SYSTEM temexdmodluyben2
  (* Version 1.0, Author, 4DIAC-Consortium *)
  APPLICATION temexdmod
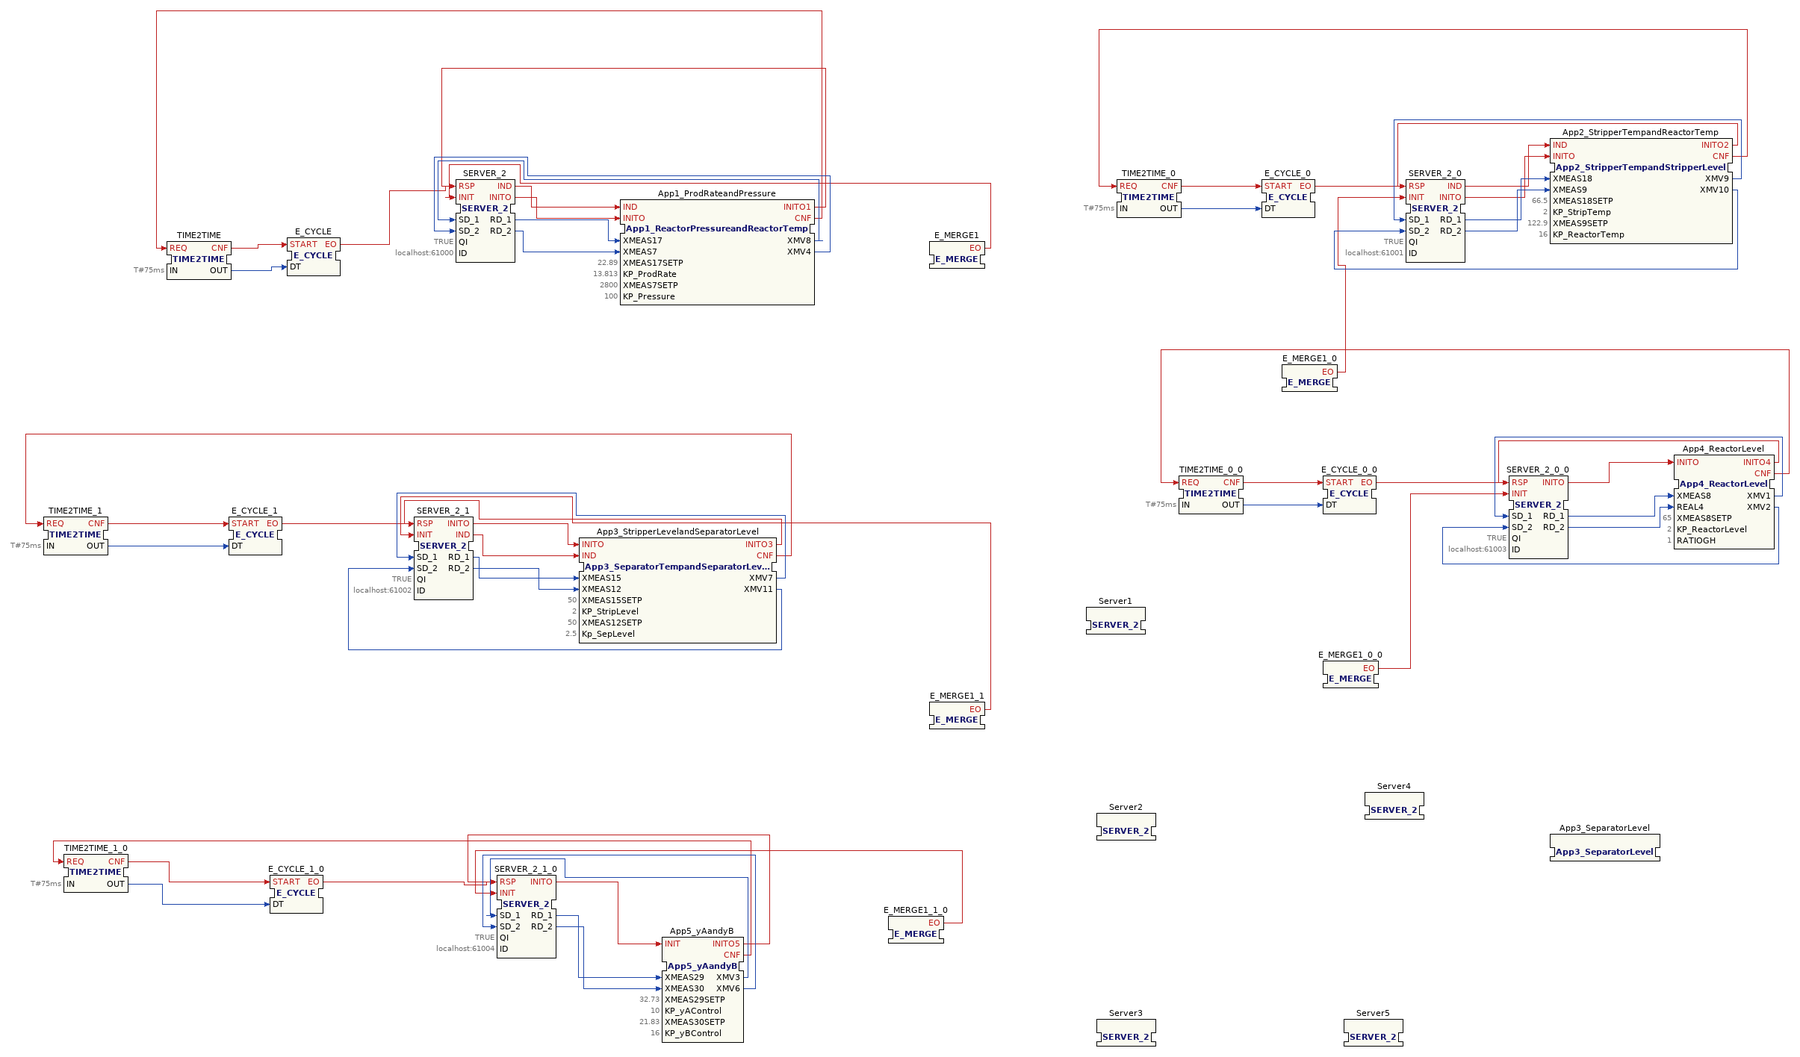
    FBS
      E_MERGE1 : E_MERGE;
      SERVER_2 : SERVER_2(QI := TRUE, ID := localhost:61000);
      TIME2TIME : TIME2TIME(IN := T#75ms);
      E_CYCLE : E_CYCLE;
      App1_ProdRateandPressure : App1_ReactorPressureandReactorTemp(XMEAS17SETP := 22.89, KP_ProdRate := 13.813, XMEAS7SETP := 2800, KP_Pressure := 100);
      TIME2TIME_0 : TIME2TIME(IN := T#75ms);
      E_CYCLE_0 : E_CYCLE;
      SERVER_2_0 : SERVER_2(QI := TRUE, ID := localhost:61001);
      E_MERGE1_0 : E_MERGE;
      App2_StripperTempandReactorTemp : App2_StripperTempandStripperLevel(XMEAS18SETP := 66.5, KP_StripTemp := 2, XMEAS9SETP := 122.9, KP_ReactorTemp := 16);
      App3_StripperLevelandSeparatorLevel : App3_SeparatorTempandSeparatorLevel(XMEAS15SETP := 50, KP_StripLevel := 2, XMEAS12SETP := 50, Kp_SepLevel := 2.5);
      SERVER_2_1 : SERVER_2(QI := TRUE, ID := localhost:61002);
      E_CYCLE_1 : E_CYCLE;
      TIME2TIME_1 : TIME2TIME(IN := T#75ms);
      E_MERGE1_1 : E_MERGE;
      App4_ReactorLevel : App4_ReactorLevel(XMEAS8SETP := 65, KP_ReactorLevel := 2, RATIOGH := 1);
      TIME2TIME_0_0 : TIME2TIME(IN := T#75ms);
      E_CYCLE_0_0 : E_CYCLE;
      SERVER_2_0_0 : SERVER_2(QI := TRUE, ID := localhost:61003);
      E_MERGE1_0_0 : E_MERGE;
      App5_yAandyB : App5_yAandyB(XMEAS29SETP := 32.73, KP_yAControl := 10, XMEAS30SETP := 21.83, KP_yBControl := 16);
      E_CYCLE_1_0 : E_CYCLE;
      SERVER_2_1_0 : SERVER_2(QI := TRUE, ID := localhost:61004);
      TIME2TIME_1_0 : TIME2TIME(IN := T#75ms);
      E_MERGE1_1_0 : E_MERGE;
      Server1 : SERVER_2;
      Server2 : SERVER_2;
      Server3 : SERVER_2;
      Server4 : SERVER_2;
      Server5 : SERVER_2;
      App3_SeparatorLevel : App3_SeparatorLevel;
    END_FBS
    EVENT_CONNECTIONS
      App1_ProdRateandPressure.INITO1 TO SERVER_2.RSP;
      SERVER_2.IND TO App1_ProdRateandPressure.IND;
      SERVER_2.INITO TO App1_ProdRateandPressure.INITO;
      TIME2TIME.CNF TO E_CYCLE.START;
      E_CYCLE.EO TO SERVER_2.RSP;
      App1_ProdRateandPressure.CNF TO TIME2TIME.REQ;
      E_MERGE1.EO TO SERVER_2.INIT;
      TIME2TIME_0.CNF TO E_CYCLE_0.START;
      E_CYCLE_0.EO TO SERVER_2_0.RSP;
      E_MERGE1_0.EO TO SERVER_2_0.INIT;
      SERVER_2_0.IND TO App2_StripperTempandReactorTemp.IND;
      SERVER_2_0.INITO TO App2_StripperTempandReactorTemp.INITO;
      App2_StripperTempandReactorTemp.INITO2 TO SERVER_2_0.RSP;
      App2_StripperTempandReactorTemp.CNF TO TIME2TIME_0.REQ;
      TIME2TIME_1.CNF TO E_CYCLE_1.START;
      E_CYCLE_1.EO TO SERVER_2_1.RSP;
      SERVER_2_1.INITO TO App3_StripperLevelandSeparatorLevel.INITO;
      SERVER_2_1.IND TO App3_StripperLevelandSeparatorLevel.IND;
      App3_StripperLevelandSeparatorLevel.INITO3 TO SERVER_2_1.RSP;
      App3_StripperLevelandSeparatorLevel.CNF TO TIME2TIME_1.REQ;
      E_MERGE1_1.EO TO SERVER_2_1.INIT;
      TIME2TIME_0_0.CNF TO E_CYCLE_0_0.START;
      E_CYCLE_0_0.EO TO SERVER_2_0_0.RSP;
      SERVER_2_0_0.INITO TO App4_ReactorLevel.INITO;
      App4_ReactorLevel.INITO4 TO SERVER_2_0_0.RSP;
      App4_ReactorLevel.CNF TO TIME2TIME_0_0.REQ;
      E_MERGE1_0_0.EO TO SERVER_2_0_0.INIT;
      SERVER_2_1_0.INITO TO App5_yAandyB.INIT;
      App5_yAandyB.INITO5 TO SERVER_2_1_0.RSP;
      App5_yAandyB.CNF TO TIME2TIME_1_0.REQ;
      TIME2TIME_1_0.CNF TO E_CYCLE_1_0.START;
      E_CYCLE_1_0.EO TO SERVER_2_1_0.RSP;
      E_MERGE1_1_0.EO TO SERVER_2_1_0.INIT;
    END_CONNECTIONS
    DATA_CONNECTIONS
      SERVER_2.RD_1 TO App1_ProdRateandPressure.XMEAS17;
      SERVER_2.RD_2 TO App1_ProdRateandPressure.XMEAS7;
      App1_ProdRateandPressure.XMV8 TO SERVER_2.SD_1;
      App1_ProdRateandPressure.XMV4 TO SERVER_2.SD_2;
      TIME2TIME.OUT TO E_CYCLE.DT;
      SERVER_2_0.RD_1 TO App2_StripperTempandReactorTemp.XMEAS18;
      SERVER_2_0.RD_2 TO App2_StripperTempandReactorTemp.XMEAS9;
      App2_StripperTempandReactorTemp.XMV9 TO SERVER_2_0.SD_1;
      App2_StripperTempandReactorTemp.XMV10 TO SERVER_2_0.SD_2;
      TIME2TIME_0.OUT TO E_CYCLE_0.DT;
      TIME2TIME_1.OUT TO E_CYCLE_1.DT;
      SERVER_2_1.RD_1 TO App3_StripperLevelandSeparatorLevel.XMEAS15;
      SERVER_2_1.RD_2 TO App3_StripperLevelandSeparatorLevel.XMEAS12;
      App3_StripperLevelandSeparatorLevel.XMV7 TO SERVER_2_1.SD_1;
      App3_StripperLevelandSeparatorLevel.XMV11 TO SERVER_2_1.SD_2;
      TIME2TIME_0_0.OUT TO E_CYCLE_0_0.DT;
      SERVER_2_0_0.RD_1 TO App4_ReactorLevel.XMEAS8;
      SERVER_2_0_0.RD_2 TO App4_ReactorLevel.REAL4;
      App4_ReactorLevel.XMV1 TO SERVER_2_0_0.SD_1;
      App4_ReactorLevel.XMV2 TO SERVER_2_0_0.SD_2;
      TIME2TIME_1_0.OUT TO E_CYCLE_1_0.DT;
      SERVER_2_1_0.RD_1 TO App5_yAandyB.XMEAS29;
      SERVER_2_1_0.RD_2 TO App5_yAandyB.XMEAS30;
      App5_yAandyB.XMV3 TO SERVER_2_1_0.SD_1;
      App5_yAandyB.XMV6 TO SERVER_2_1_0.SD_2;
    END_CONNECTIONS
  END_APPLICATION
  APPLICATION temexdmod2
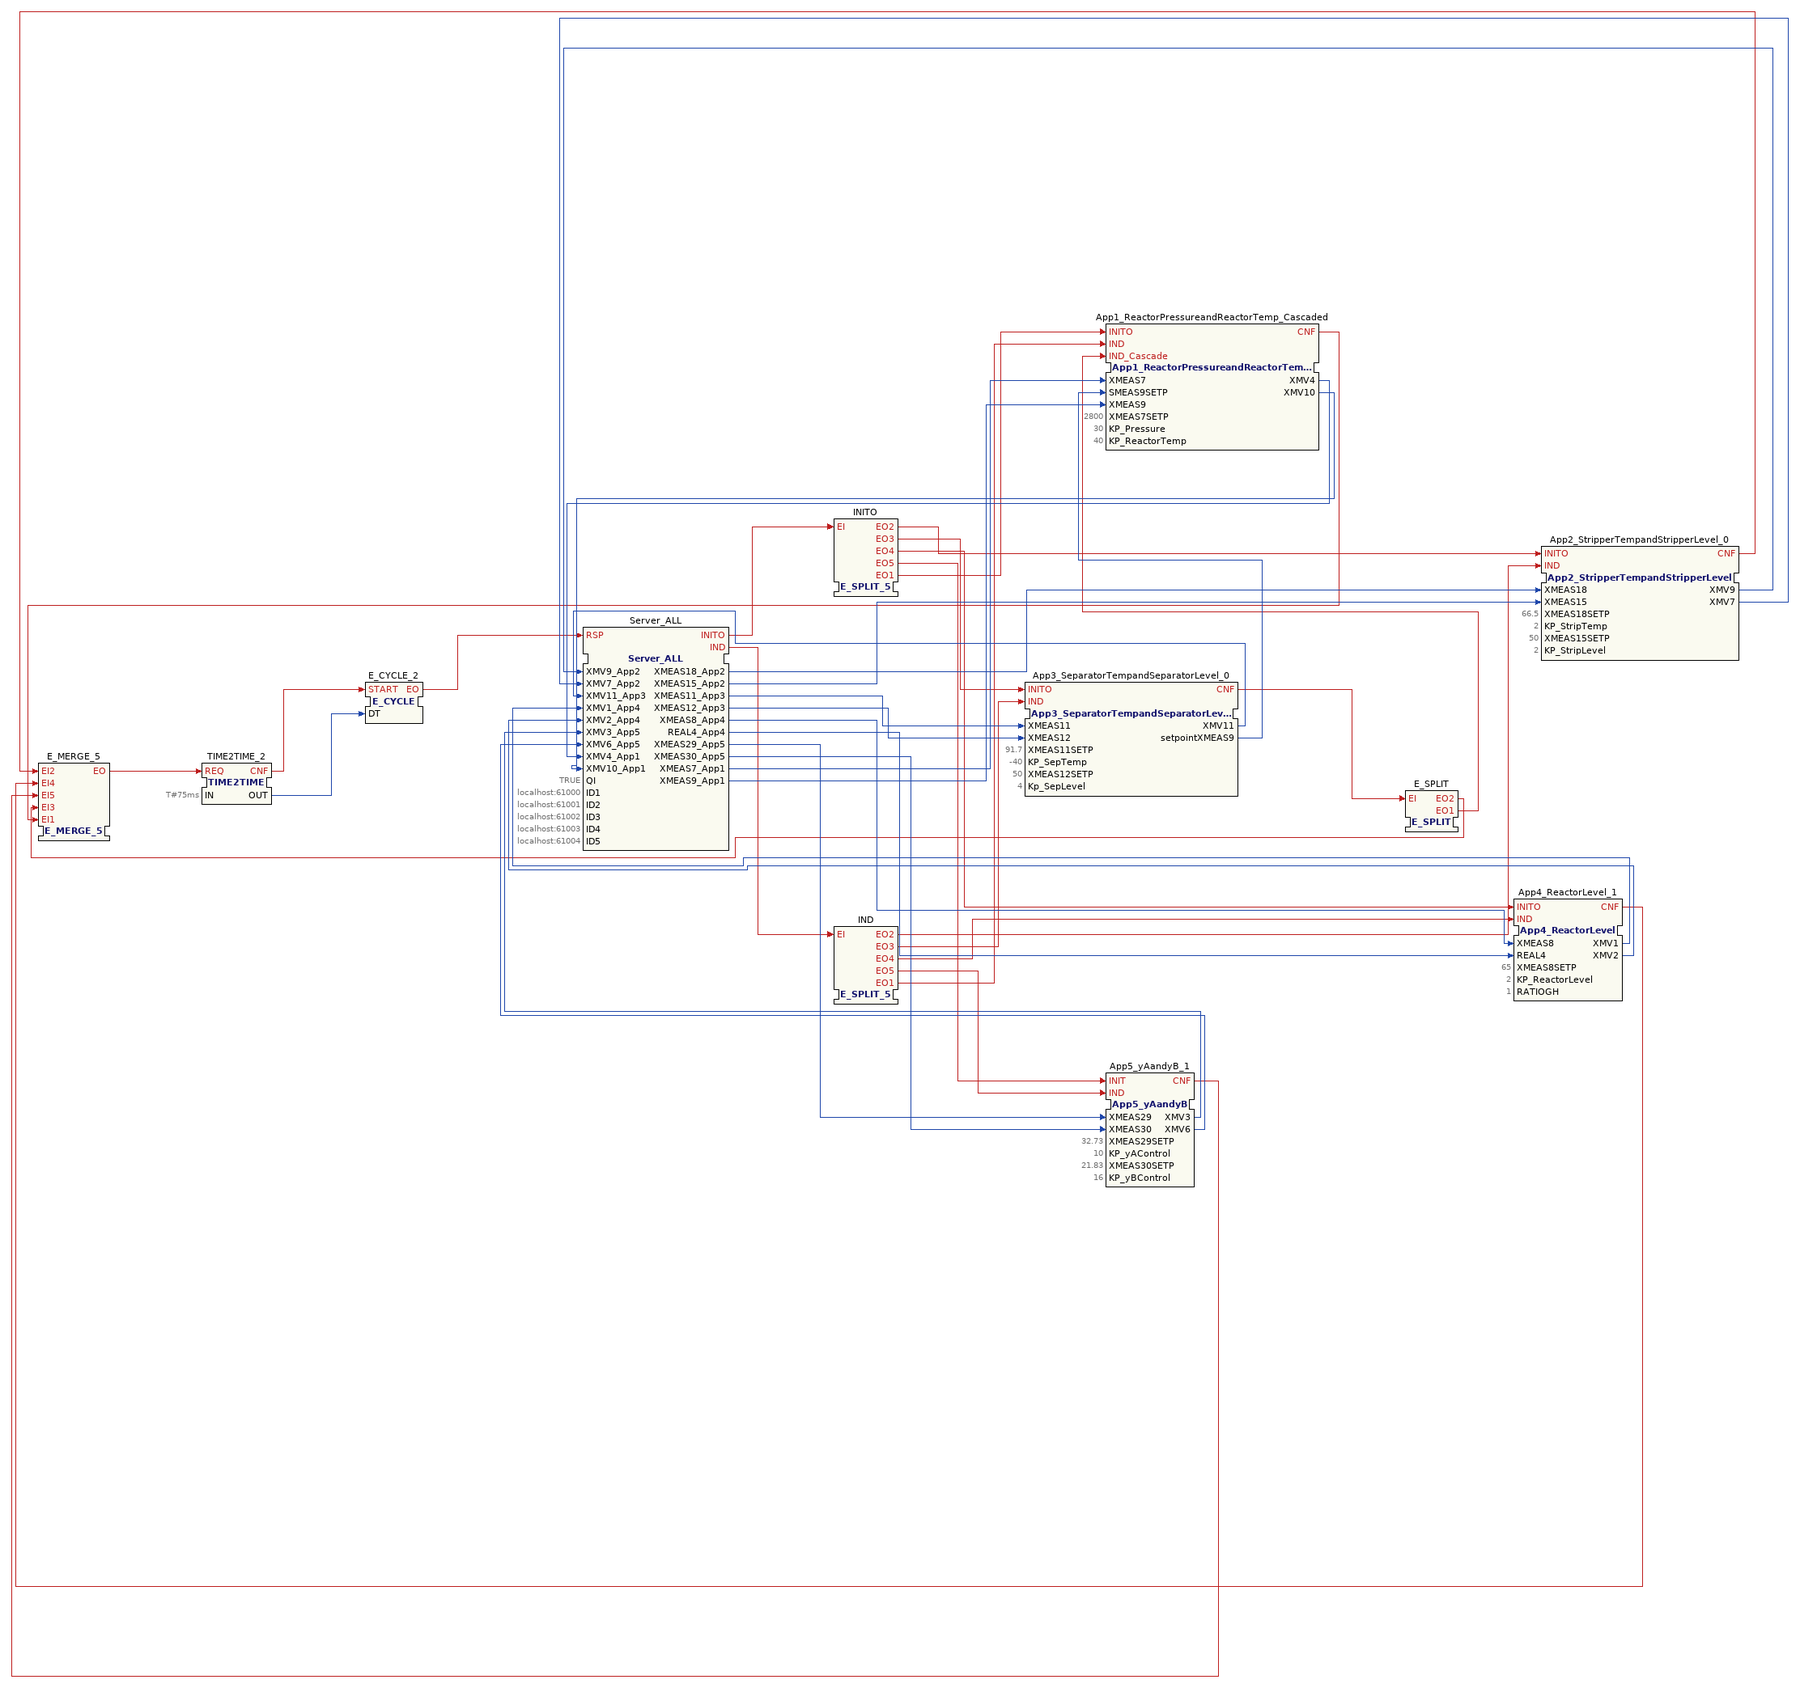
    FBS
      IND : E_SPLIT_5;
      TIME2TIME_2 : TIME2TIME(IN := T#75ms);
      E_CYCLE_2 : E_CYCLE;
      E_MERGE_5 : E_MERGE_5;
      INITO : E_SPLIT_5;
      Server_ALL : Server_ALL(QI := TRUE, ID1 := localhost:61000, ID2 := localhost:61001, ID3 := localhost:61002, ID4 := localhost:61003, ID5 := localhost:61004);
      App2_StripperTempandStripperLevel_0 : App2_StripperTempandStripperLevel(XMEAS18SETP := 66.5, KP_StripTemp := 2, XMEAS15SETP := 50, KP_StripLevel := 2);
      App3_SeparatorTempandSeparatorLevel_0 : App3_SeparatorTempandSeparatorLevel(XMEAS11SETP := 91.7, KP_SepTemp := -40, XMEAS12SETP := 50, Kp_SepLevel := 4);
      App4_ReactorLevel_1 : App4_ReactorLevel(XMEAS8SETP := 65, KP_ReactorLevel := 2, RATIOGH := 1);
      App5_yAandyB_1 : App5_yAandyB(XMEAS29SETP := 32.73, KP_yAControl := 10, XMEAS30SETP := 21.83, KP_yBControl := 16);
      App1_ReactorPressureandReactorTemp_Cascaded : App1_ReactorPressureandReactorTemp_Cascaded(XMEAS7SETP := 2800, KP_Pressure := 30, KP_ReactorTemp := 40);
      E_SPLIT : E_SPLIT;
    END_FBS
    EVENT_CONNECTIONS
      TIME2TIME_2.CNF TO E_CYCLE_2.START;
      E_MERGE_5.EO TO TIME2TIME_2.REQ;
      Server_ALL.INITO TO INITO.EI;
      Server_ALL.IND TO IND.EI;
      E_CYCLE_2.EO TO Server_ALL.RSP;
      INITO.EO2 TO App2_StripperTempandStripperLevel_0.INITO;
      INITO.EO3 TO App3_SeparatorTempandSeparatorLevel_0.INITO;
      INITO.EO4 TO App4_ReactorLevel_1.INITO;
      INITO.EO5 TO App5_yAandyB_1.INIT;
      IND.EO2 TO App2_StripperTempandStripperLevel_0.IND;
      IND.EO3 TO App3_SeparatorTempandSeparatorLevel_0.IND;
      IND.EO4 TO App4_ReactorLevel_1.IND;
      IND.EO5 TO App5_yAandyB_1.IND;
      App2_StripperTempandStripperLevel_0.CNF TO E_MERGE_5.EI2;
      App4_ReactorLevel_1.CNF TO E_MERGE_5.EI4;
      App5_yAandyB_1.CNF TO E_MERGE_5.EI5;
      INITO.EO1 TO App1_ReactorPressureandReactorTemp_Cascaded.INITO;
      IND.EO1 TO App1_ReactorPressureandReactorTemp_Cascaded.IND;
      App3_SeparatorTempandSeparatorLevel_0.CNF TO E_SPLIT.EI;
      E_SPLIT.EO2 TO E_MERGE_5.EI3;
      E_SPLIT.EO1 TO App1_ReactorPressureandReactorTemp_Cascaded.IND_Cascade;
      App1_ReactorPressureandReactorTemp_Cascaded.CNF TO E_MERGE_5.EI1;
    END_CONNECTIONS
    DATA_CONNECTIONS
      TIME2TIME_2.OUT TO E_CYCLE_2.DT;
      Server_ALL.XMEAS18_App2 TO App2_StripperTempandStripperLevel_0.XMEAS18;
      Server_ALL.XMEAS15_App2 TO App2_StripperTempandStripperLevel_0.XMEAS15;
      Server_ALL.XMEAS11_App3 TO App3_SeparatorTempandSeparatorLevel_0.XMEAS11;
      Server_ALL.XMEAS12_App3 TO App3_SeparatorTempandSeparatorLevel_0.XMEAS12;
      Server_ALL.XMEAS8_App4 TO App4_ReactorLevel_1.XMEAS8;
      Server_ALL.REAL4_App4 TO App4_ReactorLevel_1.REAL4;
      Server_ALL.XMEAS29_App5 TO App5_yAandyB_1.XMEAS29;
      Server_ALL.XMEAS30_App5 TO App5_yAandyB_1.XMEAS30;
      App2_StripperTempandStripperLevel_0.XMV9 TO Server_ALL.XMV9_App2;
      App2_StripperTempandStripperLevel_0.XMV7 TO Server_ALL.XMV7_App2;
      App3_SeparatorTempandSeparatorLevel_0.XMV11 TO Server_ALL.XMV11_App3;
      App4_ReactorLevel_1.XMV1 TO Server_ALL.XMV1_App4;
      App4_ReactorLevel_1.XMV2 TO Server_ALL.XMV2_App4;
      App5_yAandyB_1.XMV3 TO Server_ALL.XMV3_App5;
      App5_yAandyB_1.XMV6 TO Server_ALL.XMV6_App5;
      Server_ALL.XMEAS7_App1 TO App1_ReactorPressureandReactorTemp_Cascaded.XMEAS7;
      App3_SeparatorTempandSeparatorLevel_0.setpointXMEAS9 TO App1_ReactorPressureandReactorTemp_Cascaded.SMEAS9SETP;
      Server_ALL.XMEAS9_App1 TO App1_ReactorPressureandReactorTemp_Cascaded.XMEAS9;
      App1_ReactorPressureandReactorTemp_Cascaded.XMV4 TO Server_ALL.XMV4_App1;
      App1_ReactorPressureandReactorTemp_Cascaded.XMV10 TO Server_ALL.XMV10_App1;
    END_CONNECTIONS
  END_APPLICATION
  APPLICATION temexdmod3
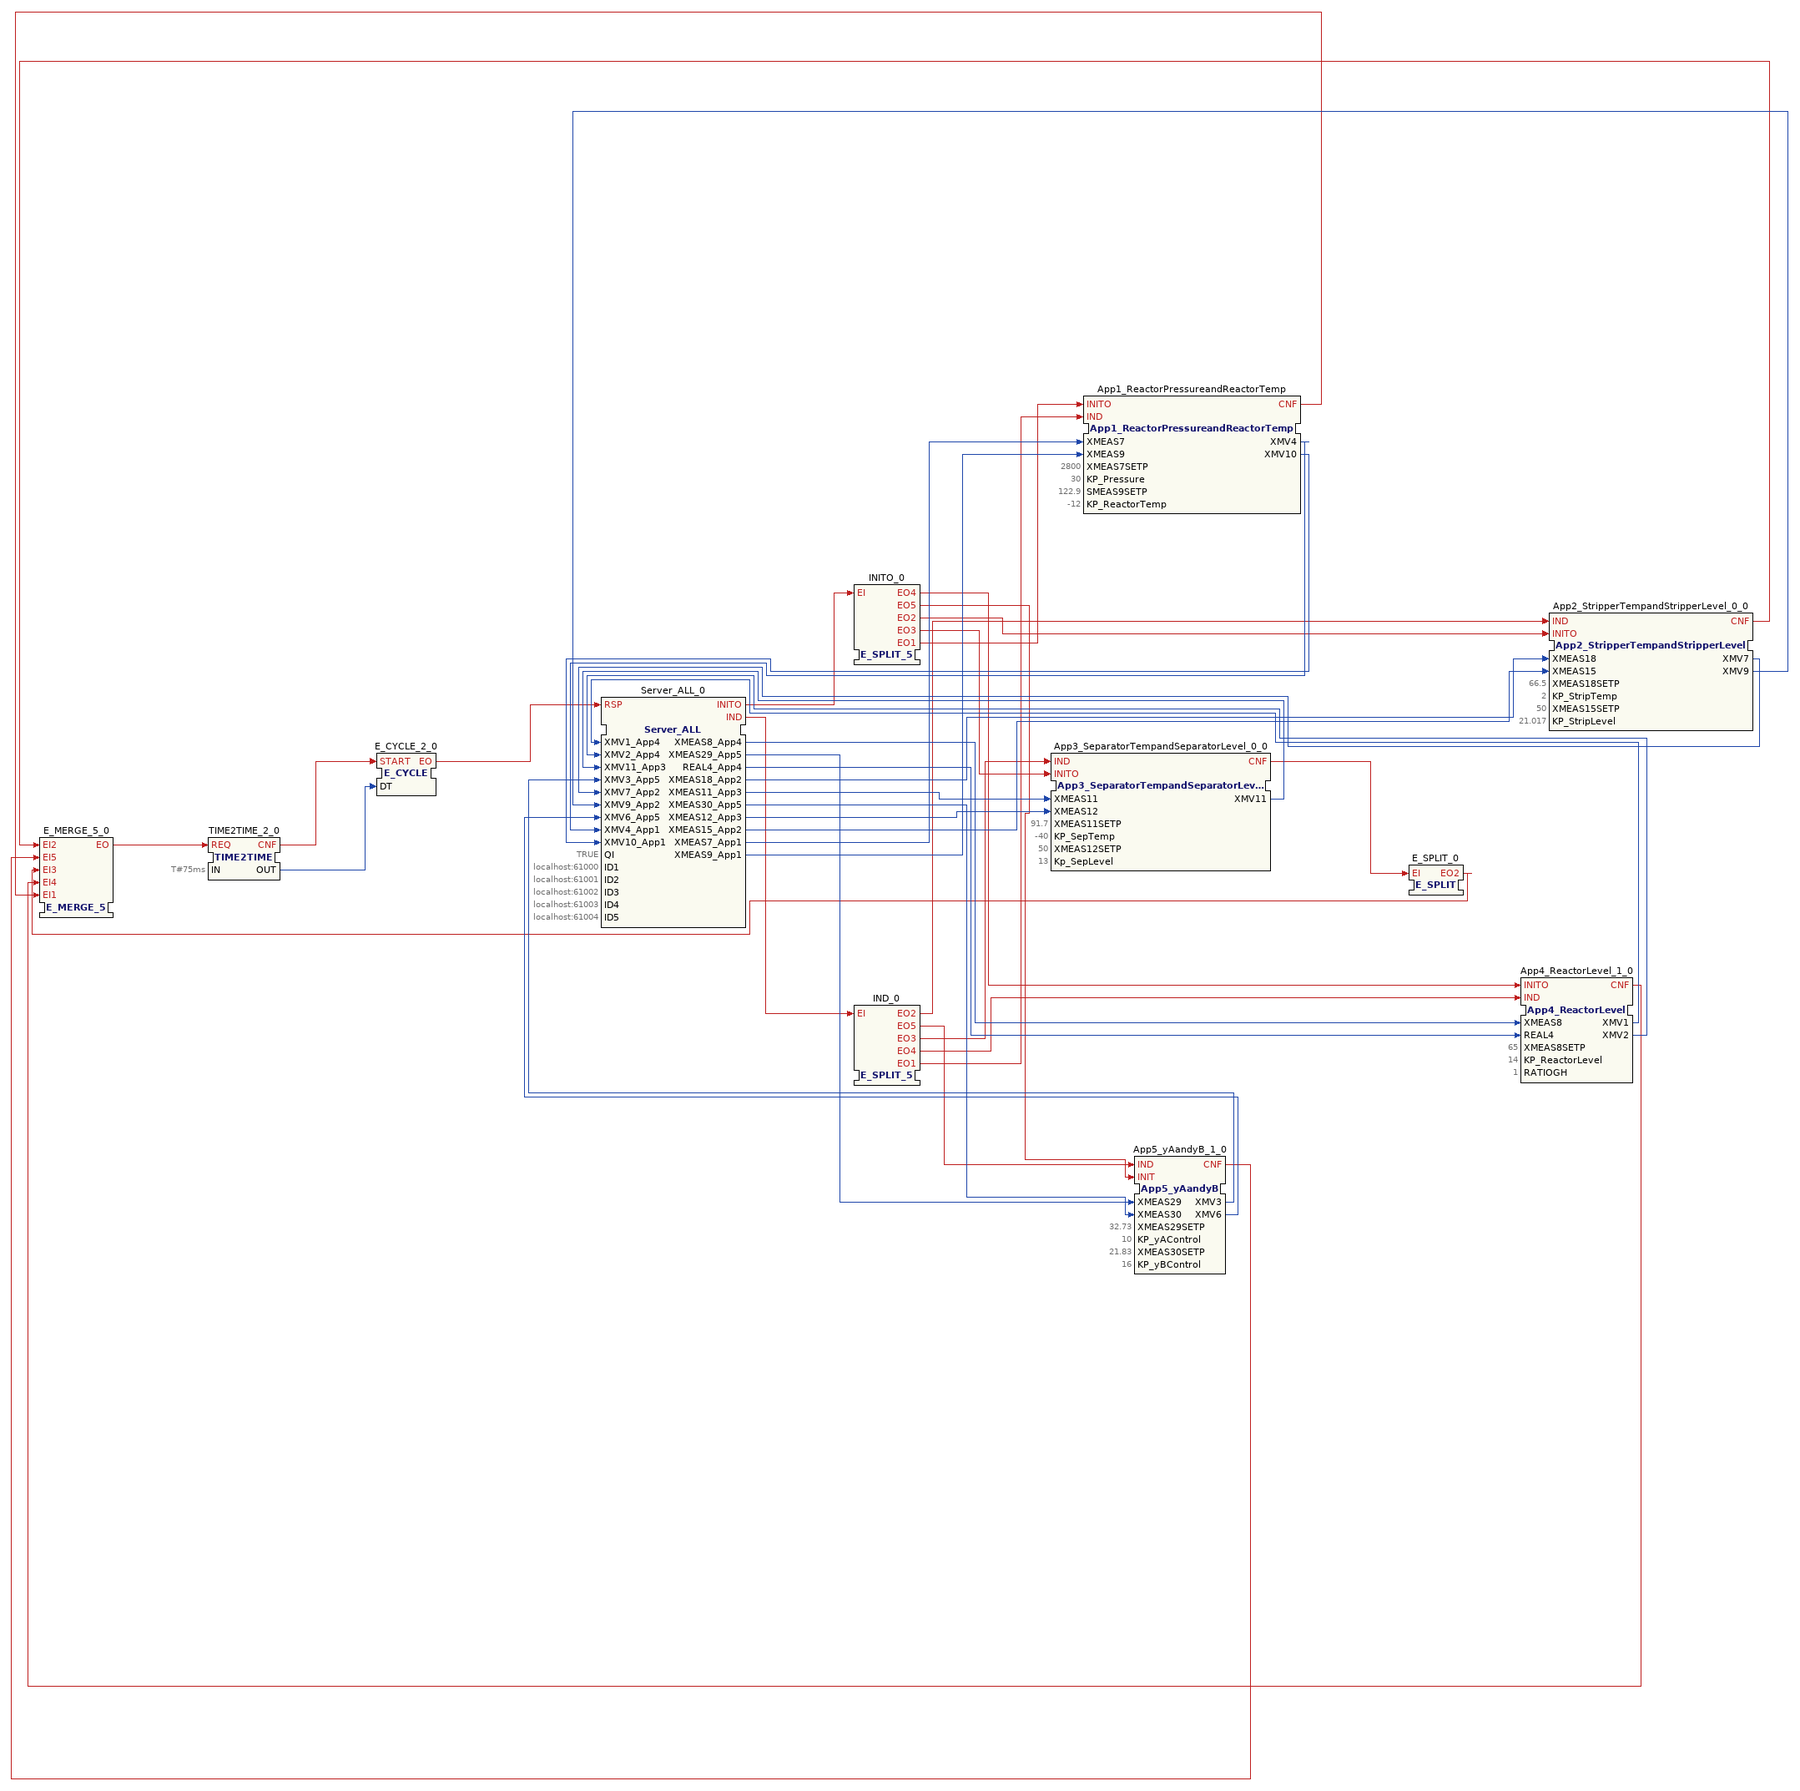
    FBS
      IND_0 : E_SPLIT_5;
      TIME2TIME_2_0 : TIME2TIME(IN := T#75ms);
      E_CYCLE_2_0 : E_CYCLE;
      E_MERGE_5_0 : E_MERGE_5;
      INITO_0 : E_SPLIT_5;
      Server_ALL_0 : Server_ALL(QI := TRUE, ID1 := localhost:61000, ID2 := localhost:61001, ID3 := localhost:61002, ID4 := localhost:61003, ID5 := localhost:61004);
      App2_StripperTempandStripperLevel_0_0 : App2_StripperTempandStripperLevel(XMEAS18SETP := 66.5, KP_StripTemp := 2, XMEAS15SETP := 50, KP_StripLevel := 21.017);
      App3_SeparatorTempandSeparatorLevel_0_0 : App3_SeparatorTempandSeparatorLevel(XMEAS11SETP := 91.7, KP_SepTemp := -40, XMEAS12SETP := 50, Kp_SepLevel := 13);
      App4_ReactorLevel_1_0 : App4_ReactorLevel(XMEAS8SETP := 65, KP_ReactorLevel := 14, RATIOGH := 1);
      App5_yAandyB_1_0 : App5_yAandyB(XMEAS29SETP := 32.73, KP_yAControl := 10, XMEAS30SETP := 21.83, KP_yBControl := 16);
      E_SPLIT_0 : E_SPLIT;
      App1_ReactorPressureandReactorTemp : App1_ReactorPressureandReactorTemp(XMEAS7SETP := 2800, KP_Pressure := 30, SMEAS9SETP := 122.9, KP_ReactorTemp := -12);
    END_FBS
    EVENT_CONNECTIONS
      IND_0.EO2 TO App2_StripperTempandStripperLevel_0_0.IND;
      App2_StripperTempandStripperLevel_0_0.CNF TO E_MERGE_5_0.EI2;
      IND_0.EO5 TO App5_yAandyB_1_0.IND;
      App5_yAandyB_1_0.CNF TO E_MERGE_5_0.EI5;
      TIME2TIME_2_0.CNF TO E_CYCLE_2_0.START;
      INITO_0.EO4 TO App4_ReactorLevel_1_0.INITO;
      INITO_0.EO5 TO App5_yAandyB_1_0.INIT;
      E_MERGE_5_0.EO TO TIME2TIME_2_0.REQ;
      E_SPLIT_0.EO2 TO E_MERGE_5_0.EI3;
      IND_0.EO3 TO App3_SeparatorTempandSeparatorLevel_0_0.IND;
      IND_0.EO4 TO App4_ReactorLevel_1_0.IND;
      App4_ReactorLevel_1_0.CNF TO E_MERGE_5_0.EI4;
      INITO_0.EO2 TO App2_StripperTempandStripperLevel_0_0.INITO;
      Server_ALL_0.INITO TO INITO_0.EI;
      E_CYCLE_2_0.EO TO Server_ALL_0.RSP;
      App3_SeparatorTempandSeparatorLevel_0_0.CNF TO E_SPLIT_0.EI;
      INITO_0.EO3 TO App3_SeparatorTempandSeparatorLevel_0_0.INITO;
      Server_ALL_0.IND TO IND_0.EI;
      INITO_0.EO1 TO App1_ReactorPressureandReactorTemp.INITO;
      IND_0.EO1 TO App1_ReactorPressureandReactorTemp.IND;
      App1_ReactorPressureandReactorTemp.CNF TO E_MERGE_5_0.EI1;
    END_CONNECTIONS
    DATA_CONNECTIONS
      App4_ReactorLevel_1_0.XMV1 TO Server_ALL_0.XMV1_App4;
      Server_ALL_0.XMEAS8_App4 TO App4_ReactorLevel_1_0.XMEAS8;
      App4_ReactorLevel_1_0.XMV2 TO Server_ALL_0.XMV2_App4;
      Server_ALL_0.XMEAS29_App5 TO App5_yAandyB_1_0.XMEAS29;
      App3_SeparatorTempandSeparatorLevel_0_0.XMV11 TO Server_ALL_0.XMV11_App3;
      TIME2TIME_2_0.OUT TO E_CYCLE_2_0.DT;
      Server_ALL_0.REAL4_App4 TO App4_ReactorLevel_1_0.REAL4;
      App5_yAandyB_1_0.XMV3 TO Server_ALL_0.XMV3_App5;
      App2_StripperTempandStripperLevel_0_0.XMV7 TO Server_ALL_0.XMV7_App2;
      Server_ALL_0.XMEAS18_App2 TO App2_StripperTempandStripperLevel_0_0.XMEAS18;
      Server_ALL_0.XMEAS11_App3 TO App3_SeparatorTempandSeparatorLevel_0_0.XMEAS11;
      Server_ALL_0.XMEAS30_App5 TO App5_yAandyB_1_0.XMEAS30;
      App2_StripperTempandStripperLevel_0_0.XMV9 TO Server_ALL_0.XMV9_App2;
      Server_ALL_0.XMEAS12_App3 TO App3_SeparatorTempandSeparatorLevel_0_0.XMEAS12;
      App5_yAandyB_1_0.XMV6 TO Server_ALL_0.XMV6_App5;
      Server_ALL_0.XMEAS15_App2 TO App2_StripperTempandStripperLevel_0_0.XMEAS15;
      Server_ALL_0.XMEAS7_App1 TO App1_ReactorPressureandReactorTemp.XMEAS7;
      Server_ALL_0.XMEAS9_App1 TO App1_ReactorPressureandReactorTemp.XMEAS9;
      App1_ReactorPressureandReactorTemp.XMV4 TO Server_ALL_0.XMV4_App1;
      App1_ReactorPressureandReactorTemp.XMV10 TO Server_ALL_0.XMV10_App1;
    END_CONNECTIONS
  END_APPLICATION
  APPLICATION temexdmod4
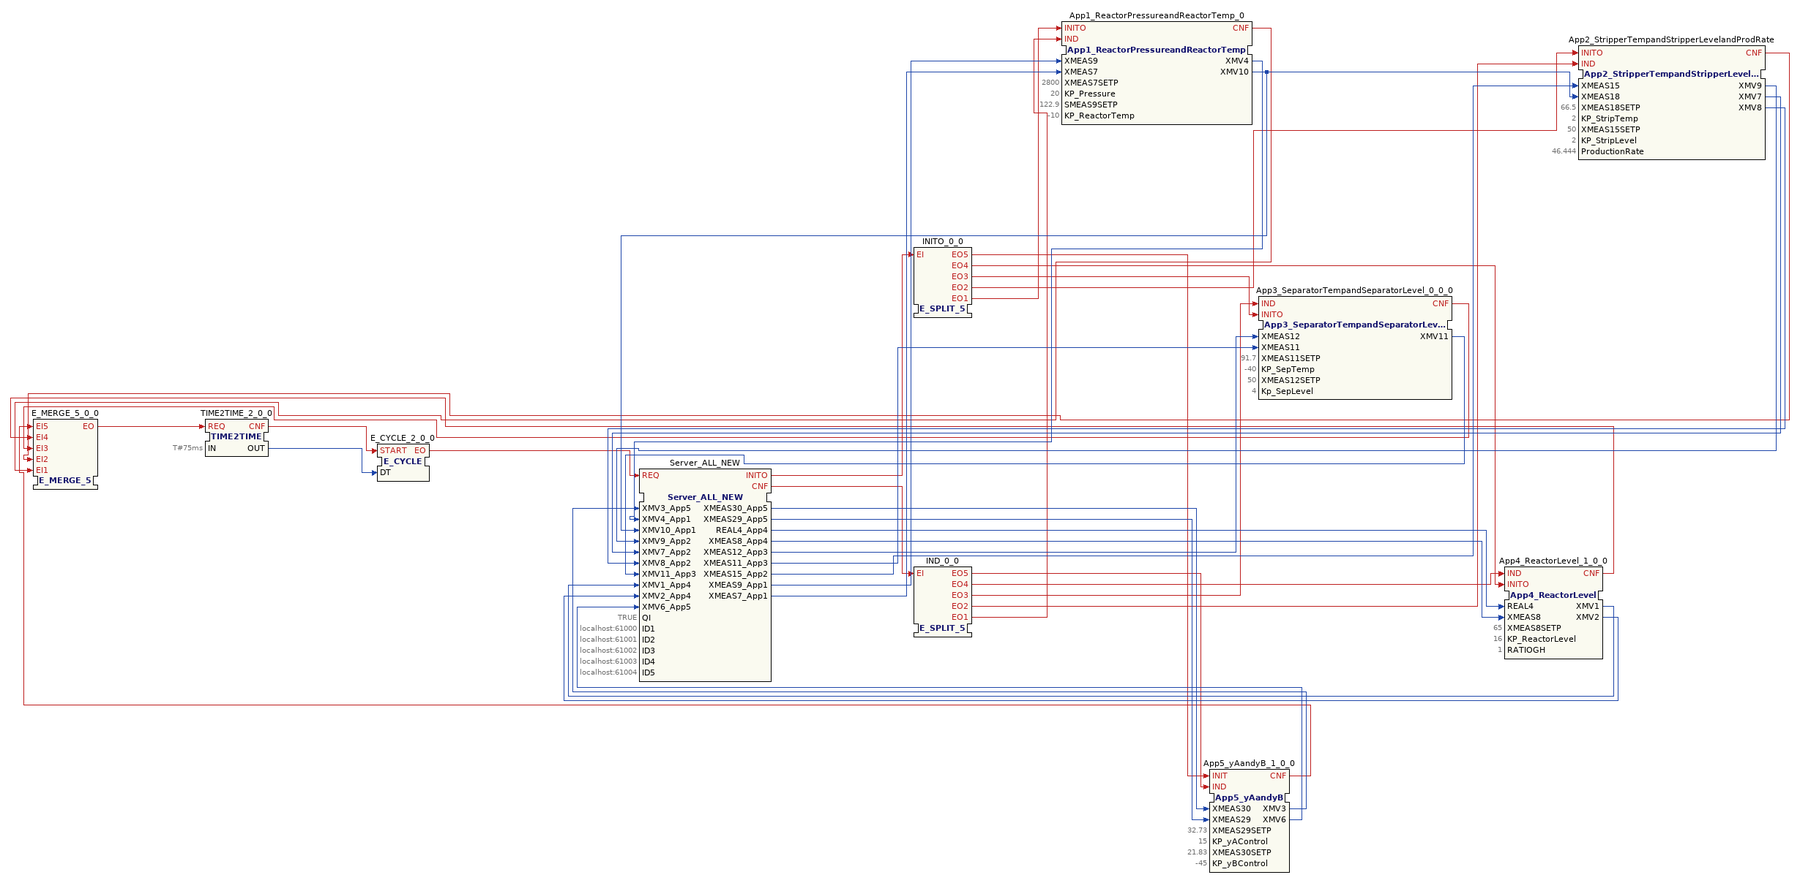
    FBS
      IND_0_0 : E_SPLIT_5;
      TIME2TIME_2_0_0 : TIME2TIME(IN := T#75ms);
      E_CYCLE_2_0_0 : E_CYCLE;
      E_MERGE_5_0_0 : E_MERGE_5;
      INITO_0_0 : E_SPLIT_5;
      App3_SeparatorTempandSeparatorLevel_0_0_0 : App3_SeparatorTempandSeparatorLevel(XMEAS11SETP := 91.7, KP_SepTemp := -40, XMEAS12SETP := 50, Kp_SepLevel := 4);
      App4_ReactorLevel_1_0_0 : App4_ReactorLevel(XMEAS8SETP := 65, KP_ReactorLevel := 16, RATIOGH := 1);
      App5_yAandyB_1_0_0 : App5_yAandyB(XMEAS29SETP := 32.73, KP_yAControl := 15, XMEAS30SETP := 21.83, KP_yBControl := -45);
      App1_ReactorPressureandReactorTemp_0 : App1_ReactorPressureandReactorTemp(XMEAS7SETP := 2800, KP_Pressure := 20, SMEAS9SETP := 122.9, KP_ReactorTemp := -10);
      App2_StripperTempandStripperLevelandProdRate : App2_StripperTempandStripperLevelandProdRate(XMEAS18SETP := 66.5, KP_StripTemp := 2, XMEAS15SETP := 50, KP_StripLevel := 2, ProductionRate := 46.444);
      Server_ALL_NEW : Server_ALL_NEW(QI := TRUE, ID1 := localhost:61000, ID2 := localhost:61001, ID3 := localhost:61002, ID4 := localhost:61003, ID5 := localhost:61004);
    END_FBS
    EVENT_CONNECTIONS
      TIME2TIME_2_0_0.CNF TO E_CYCLE_2_0_0.START;
      E_MERGE_5_0_0.EO TO TIME2TIME_2_0_0.REQ;
      INITO_0_0.EO5 TO App5_yAandyB_1_0_0.INIT;
      IND_0_0.EO5 TO App5_yAandyB_1_0_0.IND;
      App5_yAandyB_1_0_0.CNF TO E_MERGE_5_0_0.EI5;
      App4_ReactorLevel_1_0_0.CNF TO E_MERGE_5_0_0.EI4;
      App3_SeparatorTempandSeparatorLevel_0_0_0.CNF TO E_MERGE_5_0_0.EI3;
      IND_0_0.EO4 TO App4_ReactorLevel_1_0_0.IND;
      INITO_0_0.EO4 TO App4_ReactorLevel_1_0_0.INITO;
      IND_0_0.EO3 TO App3_SeparatorTempandSeparatorLevel_0_0_0.IND;
      INITO_0_0.EO3 TO App3_SeparatorTempandSeparatorLevel_0_0_0.INITO;
      App2_StripperTempandStripperLevelandProdRate.CNF TO E_MERGE_5_0_0.EI2;
      INITO_0_0.EO2 TO App2_StripperTempandStripperLevelandProdRate.INITO;
      IND_0_0.EO2 TO App2_StripperTempandStripperLevelandProdRate.IND;
      App1_ReactorPressureandReactorTemp_0.CNF TO E_MERGE_5_0_0.EI1;
      INITO_0_0.EO1 TO App1_ReactorPressureandReactorTemp_0.INITO;
      IND_0_0.EO1 TO App1_ReactorPressureandReactorTemp_0.IND;
      Server_ALL_NEW.INITO TO INITO_0_0.EI;
      Server_ALL_NEW.CNF TO IND_0_0.EI;
      E_CYCLE_2_0_0.EO TO Server_ALL_NEW.REQ;
    END_CONNECTIONS
    DATA_CONNECTIONS
      TIME2TIME_2_0_0.OUT TO E_CYCLE_2_0_0.DT;
      Server_ALL_NEW.XMEAS30_App5 TO App5_yAandyB_1_0_0.XMEAS30;
      Server_ALL_NEW.XMEAS29_App5 TO App5_yAandyB_1_0_0.XMEAS29;
      Server_ALL_NEW.REAL4_App4 TO App4_ReactorLevel_1_0_0.REAL4;
      Server_ALL_NEW.XMEAS8_App4 TO App4_ReactorLevel_1_0_0.XMEAS8;
      Server_ALL_NEW.XMEAS12_App3 TO App3_SeparatorTempandSeparatorLevel_0_0_0.XMEAS12;
      Server_ALL_NEW.XMEAS11_App3 TO App3_SeparatorTempandSeparatorLevel_0_0_0.XMEAS11;
      Server_ALL_NEW.XMEAS15_App2 TO App2_StripperTempandStripperLevelandProdRate.XMEAS15;
      Server_ALL_NEW.XMEAS9_App1 TO App1_ReactorPressureandReactorTemp_0.XMEAS9;
      Server_ALL_NEW.XMEAS7_App1 TO App1_ReactorPressureandReactorTemp_0.XMEAS7;
      App5_yAandyB_1_0_0.XMV3 TO Server_ALL_NEW.XMV3_App5;
      App1_ReactorPressureandReactorTemp_0.XMV4 TO Server_ALL_NEW.XMV4_App1;
      App1_ReactorPressureandReactorTemp_0.XMV10 TO Server_ALL_NEW.XMV10_App1;
      App2_StripperTempandStripperLevelandProdRate.XMV9 TO Server_ALL_NEW.XMV9_App2;
      App2_StripperTempandStripperLevelandProdRate.XMV7 TO Server_ALL_NEW.XMV7_App2;
      App2_StripperTempandStripperLevelandProdRate.XMV8 TO Server_ALL_NEW.XMV8_App2;
      App3_SeparatorTempandSeparatorLevel_0_0_0.XMV11 TO Server_ALL_NEW.XMV11_App3;
      App4_ReactorLevel_1_0_0.XMV1 TO Server_ALL_NEW.XMV1_App4;
      App4_ReactorLevel_1_0_0.XMV2 TO Server_ALL_NEW.XMV2_App4;
      App5_yAandyB_1_0_0.XMV6 TO Server_ALL_NEW.XMV6_App5;
      App1_ReactorPressureandReactorTemp_0.XMV10 TO App2_StripperTempandStripperLevelandProdRate.XMEAS18;
    END_CONNECTIONS
  END_APPLICATION
  DEVICE FORTE_PC : FORTE_PC(MGR_ID := "localhost:61499")
    {SET_ATTRIBUTE(Profile, HOLOBLOC)}
    RESOURCE EMB_RES : EMB_RES
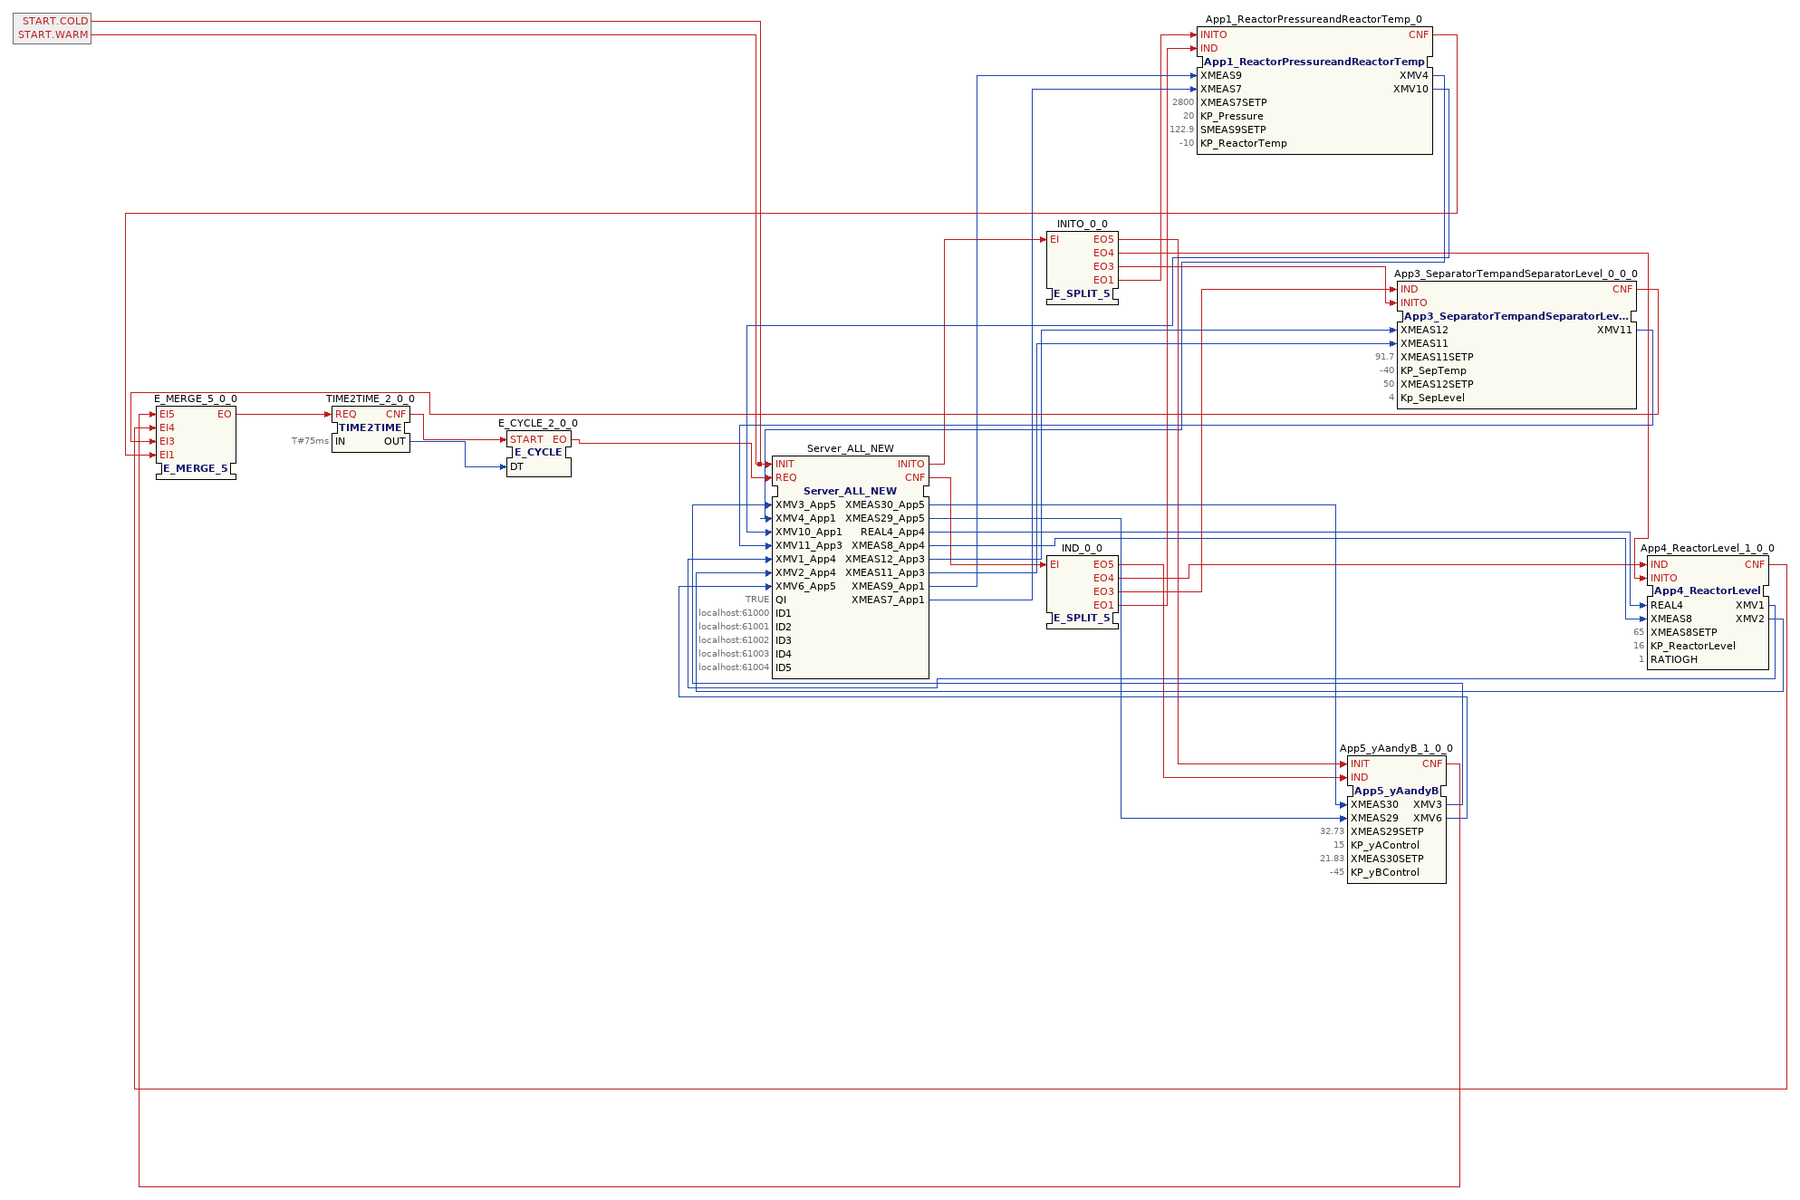
      FBS
        IND_0_0 : E_SPLIT_5;
        TIME2TIME_2_0_0 : TIME2TIME(IN := T#75ms);
        E_CYCLE_2_0_0 : E_CYCLE;
        E_MERGE_5_0_0 : E_MERGE_5;
        INITO_0_0 : E_SPLIT_5;
        App3_SeparatorTempandSeparatorLevel_0_0_0 : App3_SeparatorTempandSeparatorLevel(XMEAS11SETP := 91.7, KP_SepTemp := -40, XMEAS12SETP := 50, Kp_SepLevel := 4);
        App4_ReactorLevel_1_0_0 : App4_ReactorLevel(XMEAS8SETP := 65, KP_ReactorLevel := 16, RATIOGH := 1);
        App5_yAandyB_1_0_0 : App5_yAandyB(XMEAS29SETP := 32.73, KP_yAControl := 15, XMEAS30SETP := 21.83, KP_yBControl := -45);
        App1_ReactorPressureandReactorTemp_0 : App1_ReactorPressureandReactorTemp(XMEAS7SETP := 2800, KP_Pressure := 20, SMEAS9SETP := 122.9, KP_ReactorTemp := -10);
        Server_ALL_NEW : Server_ALL_NEW(QI := TRUE, ID1 := localhost:61000, ID2 := localhost:61001, ID3 := localhost:61002, ID4 := localhost:61003, ID5 := localhost:61004);
      END_FBS
      EVENT_CONNECTIONS
        TIME2TIME_2_0_0.CNF TO E_CYCLE_2_0_0.START;
        START.COLD TO Server_ALL_NEW.INIT;
        START.WARM TO Server_ALL_NEW.INIT;
        E_MERGE_5_0_0.EO TO TIME2TIME_2_0_0.REQ;
        INITO_0_0.EO5 TO App5_yAandyB_1_0_0.INIT;
        IND_0_0.EO5 TO App5_yAandyB_1_0_0.IND;
        App5_yAandyB_1_0_0.CNF TO E_MERGE_5_0_0.EI5;
        App4_ReactorLevel_1_0_0.CNF TO E_MERGE_5_0_0.EI4;
        App3_SeparatorTempandSeparatorLevel_0_0_0.CNF TO E_MERGE_5_0_0.EI3;
        IND_0_0.EO4 TO App4_ReactorLevel_1_0_0.IND;
        INITO_0_0.EO4 TO App4_ReactorLevel_1_0_0.INITO;
        IND_0_0.EO3 TO App3_SeparatorTempandSeparatorLevel_0_0_0.IND;
        INITO_0_0.EO3 TO App3_SeparatorTempandSeparatorLevel_0_0_0.INITO;
        App1_ReactorPressureandReactorTemp_0.CNF TO E_MERGE_5_0_0.EI1;
        INITO_0_0.EO1 TO App1_ReactorPressureandReactorTemp_0.INITO;
        IND_0_0.EO1 TO App1_ReactorPressureandReactorTemp_0.IND;
        Server_ALL_NEW.INITO TO INITO_0_0.EI;
        Server_ALL_NEW.CNF TO IND_0_0.EI;
        E_CYCLE_2_0_0.EO TO Server_ALL_NEW.REQ;
      END_CONNECTIONS
      DATA_CONNECTIONS
        TIME2TIME_2_0_0.OUT TO E_CYCLE_2_0_0.DT;
        Server_ALL_NEW.XMEAS30_App5 TO App5_yAandyB_1_0_0.XMEAS30;
        Server_ALL_NEW.XMEAS29_App5 TO App5_yAandyB_1_0_0.XMEAS29;
        Server_ALL_NEW.REAL4_App4 TO App4_ReactorLevel_1_0_0.REAL4;
        Server_ALL_NEW.XMEAS8_App4 TO App4_ReactorLevel_1_0_0.XMEAS8;
        Server_ALL_NEW.XMEAS12_App3 TO App3_SeparatorTempandSeparatorLevel_0_0_0.XMEAS12;
        Server_ALL_NEW.XMEAS11_App3 TO App3_SeparatorTempandSeparatorLevel_0_0_0.XMEAS11;
        Server_ALL_NEW.XMEAS9_App1 TO App1_ReactorPressureandReactorTemp_0.XMEAS9;
        Server_ALL_NEW.XMEAS7_App1 TO App1_ReactorPressureandReactorTemp_0.XMEAS7;
        App5_yAandyB_1_0_0.XMV3 TO Server_ALL_NEW.XMV3_App5;
        App1_ReactorPressureandReactorTemp_0.XMV4 TO Server_ALL_NEW.XMV4_App1;
        App1_ReactorPressureandReactorTemp_0.XMV10 TO Server_ALL_NEW.XMV10_App1;
        App3_SeparatorTempandSeparatorLevel_0_0_0.XMV11 TO Server_ALL_NEW.XMV11_App3;
        App4_ReactorLevel_1_0_0.XMV1 TO Server_ALL_NEW.XMV1_App4;
        App4_ReactorLevel_1_0_0.XMV2 TO Server_ALL_NEW.XMV2_App4;
        App5_yAandyB_1_0_0.XMV6 TO Server_ALL_NEW.XMV6_App5;
      END_CONNECTIONS
    END_RESOURCE
  END_DEVICE
  MAPPINGS
    temexdmod4.IND_0_0 ON FORTE_PC.EMB_RES.IND_0_0;
    temexdmod4.TIME2TIME_2_0_0 ON FORTE_PC.EMB_RES.TIME2TIME_2_0_0;
    temexdmod4.E_CYCLE_2_0_0 ON FORTE_PC.EMB_RES.E_CYCLE_2_0_0;
    temexdmod4.E_MERGE_5_0_0 ON FORTE_PC.EMB_RES.E_MERGE_5_0_0;
    temexdmod4.INITO_0_0 ON FORTE_PC.EMB_RES.INITO_0_0;
    temexdmod4.App3_SeparatorTempandSeparatorLevel_0_0_0 ON FORTE_PC.EMB_RES.App3_SeparatorTempandSeparatorLevel_0_0_0;
    temexdmod4.App4_ReactorLevel_1_0_0 ON FORTE_PC.EMB_RES.App4_ReactorLevel_1_0_0;
    temexdmod4.App5_yAandyB_1_0_0 ON FORTE_PC.EMB_RES.App5_yAandyB_1_0_0;
    temexdmod4.App1_ReactorPressureandReactorTemp_0 ON FORTE_PC.EMB_RES.App1_ReactorPressureandReactorTemp_0;
    temexdmod4.Server_ALL_NEW ON FORTE_PC.EMB_RES.Server_ALL_NEW;
  END_MAPPINGS
  SEGMENTS
    Ethernet : Ethernet;
  END_SEGMENTS
  LINKS
    FORTE_PC => Ethernet;
  END_LINKS
END_SYSTEM
